Yaskawa INFORM job: JUMPTRC.JBI

/JOB
//NAME JUMPTRC
//POS
///NPOS 20,0,0,0,0,0
///TOOL 0
///POSTYPE PULSE
///PULSE
C00000=-2822,58859,-1118,-1041,-34109,-89
C00001=-2161,58790,-1247,-1129,-34038,-353
C00002=-2445,58630,-1496,-1095,-33938,-237
C00003=-2689,58371,-1892,-1067,-33780,-136
C00004=-2833,58024,-2418,-1053,-33569,-74
C00005=-2882,57620,-3027,-1052,-33325,-50
C00006=-2836,57220,-3630,-1064,-33082,-63
C00007=-2687,56867,-4161,-1090,-32868,-119
C00008=-2427,56622,-4532,-1128,-32716,-220
C00009=-2127,56487,-4736,-1171,-32630,-337
C00010=-1792,56495,-4724,-1216,-32632,-471
C00011=-1504,56651,-4486,-1252,-32725,-588
C00012=-1257,56923,-4071,-1281,-32891,-691
C00013=-1112,57266,-3548,-1294,-33103,-754
C00014=-1067,57664,-2940,-1293,-33350,-778
C00015=-1132,58052,-2348,-1277,-33590,-757
C00016=-1284,58402,-1818,-1251,-33806,-701
C00017=-1544,58646,-1452,-1212,-33955,-600
C00018=-1822,58769,-1271,-1174,-34028,-490
C00019=-2161,58790,-1247,-1129,-34038,-353
//INST
///DATE 2026/04/15 15:34
///ATTR SC,RW
///GROUP1 RB1
NOP
MOVJ C00000 VJ=0.78
MOVJ C00001 VJ=0.78
MOVL C00002 V=20.0
MOVL C00003 V=20.0
MOVL C00004 V=20.0
MOVL C00005 V=20.0
MOVL C00006 V=20.0
MOVL C00007 V=20.0
MOVL C00008 V=20.0
MOVL C00009 V=20.0
MOVL C00010 V=20.0
MOVL C00011 V=20.0
MOVL C00012 V=20.0
MOVL C00013 V=20.0
MOVL C00014 V=20.0
MOVL C00015 V=20.0
MOVL C00016 V=20.0
MOVL C00017 V=20.0
MOVL C00018 V=20.0
MOVL C00019 V=20.0
END
